FUNCTION_BLOCK FB_MoveBezier
VAR_INPUT
END_VAR
VAR_OUTPUT
END_VAR
VAR
END_VAR

END_FUNCTION_BLOCK

(* stored: Version 1.1.0.1, ProductVersion 3.1.4022.18
   POU FB_MoveBezier: Id {5c057fcb-a0c1-45a6-87bf-aeff6129ee29}, SpecialFunc None *)
